// TwinCAT 3 PLC project PLC_code
// ProgramVersion: 3.1.4022.4
// libraries:
//   Tc2_EnOcean, * (Beckhoff Automation GmbH)
//   Tc2_Standard, * (Beckhoff Automation GmbH)
//   Tc2_System, * (Beckhoff Automation GmbH)
//   Tc3_Module, * (Beckhoff Automation GmbH)
//   VisuSymbols,3.5.10.0,System
// project tree:
//   / GlobalTextList.TcGTLO, PlcTask.TcTTO, Visualization Manager.TcVMO (not stored)
//   GVLs/ IO.TcGVL
//   POUs/ EnOcean.TcPOU, MAIN.TcPOU, SearchEnOcean.TcPOU, SwitchEnOcean.TcPOU
//   VISUs/ Visualization.TcVIS
// real-time tasks:
//   TASK PlcTask: cycle T#10ms, priority 20, ADS port 350
// I/O:
//   DEVICE Device 1 (EtherCAT), AmsNetId 5.29.55.234.2.1
//     Term 1 (EK1100) [EK1100 EtherCAT Coupler (2A E-Bus)]
//       Term 2 (EL1008) [EL1008 8Ch. Dig. Input 24V, 3ms]
//       Term 3 (EL1008) [EL1008 8Ch. Dig. Input 24V, 3ms]
//       Term 4 (EL2008) [EL2008 8Ch. Dig. Output 24V, 0.5A]
//       Term 5 (EL2008) [EL2008 8Ch. Dig. Output 24V, 0.5A]
//       Term 6 (EL3002) [EL3002 2Ch. Ana. Input +/-10V]
//       Term 7 (EL4002) [EL4002 2Ch. Ana. Output 0-10V, 12bit]
//       Term 8 (EL3124) [EL3124 4Ch. Ana. Input 4-20mA Diff.]
//       Term 9 (EL4024) [EL4024 4Ch. Ana. Output 4-20mA, 12bit]
//       Box 10 (BK1250)
//   DEVICE Device 3 (EtherCAT Automation Protocol) (disabled), AmsNetId 5.29.55.234.4.1
// variable links:
//   PLC_code/PLC_code Instance <-> Device 1 (EtherCAT)/Term 1 (EK1100)/Box 10 (BK1250)
//     PlcTask Inputs/IO.stKL6581_In/CNODE <-> Term 2 (KL6581)/Channel 1/Input CNODE
//     PlcTask Inputs/IO.stKL6581_In/DB{0..3} <-> Term 2 (KL6581)/Channel 1/Input DB{0..3}  (4 links)
//     PlcTask Inputs/IO.stKL6581_In/ID{0..3} <-> Term 2 (KL6581)/Channel 1/Input ID{0..3}  (4 links)
//     PlcTask Inputs/IO.stKL6581_In/ORG <-> Term 2 (KL6581)/Channel 1/Input ORG
//     PlcTask Inputs/IO.stKL6581_In/STATUS <-> Term 2 (KL6581)/Channel 1/Input STATUS
//     PlcTask Inputs/IO.stKL6581_In/nStatus <-> Term 2 (KL6581)/Channel 1/Status
//     PlcTask Outputs/IO.stKL6581_Out/CNODE <-> Term 2 (KL6581)/Channel 1/Output CNODE
//     PlcTask Outputs/IO.stKL6581_Out/DB{0..3} <-> Term 2 (KL6581)/Channel 1/Output DB{0..3}  (4 links)
//     PlcTask Outputs/IO.stKL6581_Out/ID{0..3} <-> Term 2 (KL6581)/Channel 1/Output ID{0..3}  (4 links)
//     PlcTask Outputs/IO.stKL6581_Out/ORG <-> Term 2 (KL6581)/Channel 1/Output ORG
//     PlcTask Outputs/IO.stKL6581_Out/STATUS <-> Term 2 (KL6581)/Channel 1/Output STATUS
//     PlcTask Outputs/IO.stKL6581_Out/nControl <-> Term 2 (KL6581)/Channel 1/Control

CONFIGURATION PLC_code
    RESOURCE PLC ON TwinCAT3
        TASK PlcTask(INTERVAL := T#10ms, PRIORITY := 20);
        PROGRAM MAIN WITH PlcTask : MAIN;
    END_RESOURCE
END_CONFIGURATION

// ---- GVLs/IO.TcGVL
{attribute 'qualified_only'}
VAR_GLOBAL
	stKL6581_In AT %I*: KL6581_Input;
	stKL6581_Out AT %Q*: KL6581_Output;
	str_KL6581: STR_KL6581;
	//devices_id: ARRAY [0..255] OF DWORD;
END_VAR

// ---- POUs/MAIN.TcPOU
PROGRAM MAIN
VAR;
	InitEnOcean: EnOCean;
	Switches: SwitchEnOcean;
	Search: SearchEnOcean;
END_VAR

InitEnOcean();
Switches();
Search();

END_PROGRAM

// ---- POUs/EnOcean.TcPOU
FUNCTION_BLOCK EnOcean
VAR_INPUT
END_VAR
VAR_OUTPUT
END_VAR
VAR
	EnOceanRev: FB_KL6581;
	bReady: BOOL;
	bBusy: BOOL;
	bError: BOOL;
	iErrorID: INT;
END_VAR

//Initialize EnOcean gateway
EnOceanRev(
	bInit:= TRUE, 
	nIdx:= 1, 
	bReady=> bReady, 
	bBusy=> bBusy, 
	bError=> bError, 
	iErrorID=> iErrorID, 
	str_KL6581=> IO.str_KL6581, 
	stKL6581_in:= IO.stKL6581_In, 
	stKL6581_out:= IO.stKL6581_Out);

END_FUNCTION_BLOCK

// ---- POUs/SwitchEnOcean.TcPOU
FUNCTION_BLOCK SwitchEnOcean
VAR_INPUT
END_VAR
VAR_OUTPUT
END_VAR
VAR
	SwitchEnOcean: FB_Rec_RPS_Switch;
	byNode: BYTE;
	dw_ID: DWORD;
	bReceive: BOOL;
	outNode: BYTE;
	str_EnOceanSwitch: STR_EnOceanSwitch;
END_VAR

//Listening for switch EnOcean
byNode := 0;
dw_ID := 2943328; //ID of switch, need to searched 
SwitchEnOcean(
	str_KL6581:= IO.str_KL6581, 
	byNode:= byNode, 
	dw_ID:= dw_ID, 
	str_EnOceanSwitch=> str_EnOceanSwitch, 
	by_Node=> outNode, 
	bReceive=> bReceive);

END_FUNCTION_BLOCK

// ---- POUs/SearchEnOcean.TcPOU
FUNCTION_BLOCK SearchEnOcean
VAR_INPUT
END_VAR
VAR_OUTPUT
END_VAR
VAR
	EnOceanSearch: FB_EnOcean_Search;
	byNode: BYTE;
	bReceive: BOOL;
	ar_ID: ARRAY [0..255] OF DWORD;
	iDevices: INT;
END_VAR

//Search and get EnOcean IDs
EnOceanSearch(
	bStart:= TRUE, 
	str_KL6581:= IO.str_KL6581, 
	byNode:= byNode, 
	bReceive=> bReceive, 
	iDevices=> iDevices, 
	ar_ID=> ar_ID);

END_FUNCTION_BLOCK

// ---- VISUs/Visualization.TcVIS
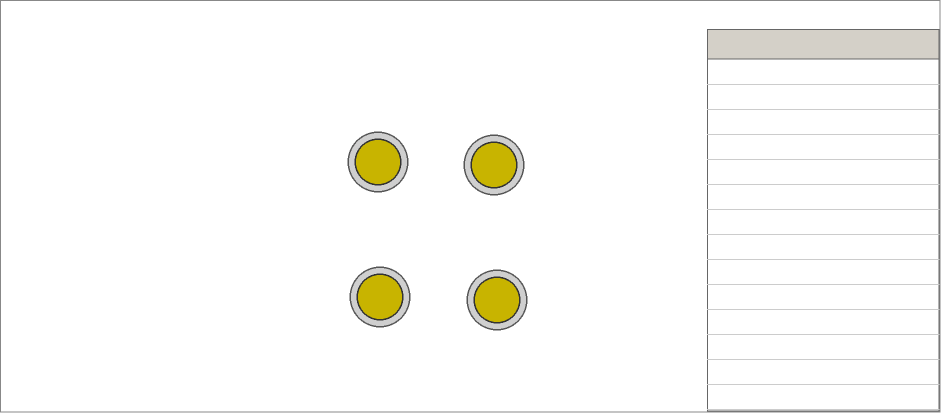
VISUALIZATION Visualization  // 941x413
    Lamp1 (459,130 70x70), variable: MAIN.Switches.str_EnOceanSwitch.bT1_ON, style: Lamp-Lamp1-Yellow
    Lamp1 (345,262 70x70), variable: MAIN.Switches.str_EnOceanSwitch.bT2_ON, style: Lamp-Lamp1-Yellow
    Lamp1 (343,127 70x70), variable: MAIN.Switches.str_EnOceanSwitch.bT1_OFF, style: Lamp-Lamp1-Yellow
    Lamp1 (462,265 70x70), variable: MAIN.Switches.str_EnOceanSwitch.bT2_OFF, style: Lamp-Lamp1-Yellow
    Table (707,29 232x382), data array: MAIN.Search.ar_ID
        p1892666644: MAIN.Search.byNode
        p338671338: MAIN.Search.bReceive
        p2170511999: MAIN.Search.ar_ID
        p3723444502: MAIN.Search.iDevices
        p3854506369: MAIN.Search.ar_ID[INDEX]
END_VISUALIZATION
